// TIA Portal V17 export
// export: Created 2025-08-13T10:43:39.5511317Z, ExportSetting WithDefaults, DisplayName Totally Integrated Automation Portal, DisplayVersion V17 Update 8, DisplayName TIA Portal Openness, DisplayVersion V17 Update 8, DisplayName TIA Portal Version Control Interface, DisplayVersion V17, DisplayName SINAMICS Startdrive Advanced, DisplayVersion V17 SP2, DisplayName SINAMICS Startdrive G110M, G120, G120C, G120D, G120P, G115D, DisplayVersion V17 SP2, DisplayName SINAMICS Startdrive G130, G150, S120, S150, SINAMICS MV, S210, DisplayVersion V17 SP2, DisplayName STEP 7 Professional, DisplayVersion V17 Update 8, DisplayName STEP 7 Safety, DisplayVersion V17 Update 6, DisplayName WinCC Advanced, DisplayVersion V17 Update 8
VAR_GLOBAL   // PLC tag table "Constants"
END_VAR
VAR_GLOBAL CONSTANT   // user constants
   LASERCOMM_LDD_ARRAY_SIZE : Int := 100;   // Size of LDD Array Data Sizes. This is for Results, DDO and Weld Mask. Tied to the number of jobs in the LDD Sequence.
   LASERCOMM_NUMBER_OF_LASERS : Int := 1;   // Number of Lasers systems on Cell
   LASERCOMM_REF_PLANE : DInt := 12345;   // LDD Reference Plane Position
END_VAR
